// TwinCAT 3 PLC project Sample_Delivery
// ProgramVersion: 3.1.4023.0
// libraries:
//   lcls-twincat-sample-delivery, * (SLAC)
//   Tc2_Standard, * (Beckhoff Automation GmbH)
//   Tc2_System, * (Beckhoff Automation GmbH)
//   Tc3_Module, * (Beckhoff Automation GmbH)
// project tree:
//   / PlcTask.TcTTO
//   POUs/ MAIN.TcPOU
// real-time tasks:
//   TASK PlcTask: cycle T#10ms, priority 20, ADS port 350
// I/O:
//   DEVICE Device 1 (EtherCAT), AmsNetId 172.21.38.26.2.1
//     Term 1 (EK1200)
//     Box 3 (EP9128-0021) [EP9128-0021 8x EtherCAT junction]
//       Term 4 (EP9128-1021) [EP9128-1021 8x EtherCAT junction - Dev A]
//       Term 5 (EP9128-2021) [EP9128-2021 8x EtherCAT junction - Dev B]
//         Box 6 (EP1111)
//         M3 Selector A Digital IO (EP2338-1001)
//         M3 Selector A Serial IO (EP6002-0002)
// variable links:
//   Sample-Delivery Instance <-> Device 1 (EtherCAT)/Box 3 (EP9128-0021)/Term 5 (EP9128-2021)/M3 Selector A Digital IO (EP2338-1001)
//     PlcTask Outputs/MAIN.fbSelectorA.stShaker01.q_xPwrDO <-> Channel 9/Output
//     PlcTask Outputs/MAIN.fbSelectorA.stShaker02.q_xPwrDO <-> Channel 10/Output
//     PlcTask Outputs/MAIN.fbSelectorA.stShaker03.q_xPwrDO <-> Channel 11/Output
//     PlcTask Outputs/MAIN.fbSelectorA.stShaker04.q_xPwrDO <-> Channel 12/Output
//   Sample-Delivery Instance <-> Device 1 (EtherCAT)/Box 3 (EP9128-0021)/Term 5 (EP9128-2021)/M3 Selector A Serial IO (EP6002-0002)
//     PlcTask Inputs/MAIN.fbSelectorA.stSensSerial.stComIn/Status <-> COM TxPDO-Map Inputs Channel 1/Status
//     PlcTask Inputs/MAIN.fbSelectorA.stViciSerial.stComIn/Status <-> COM TxPDO-Map Inputs Channel 2/Status
//     PlcTask Outputs/MAIN.fbSelectorA.stSensSerial.stComOut/Ctrl <-> COM RxPDO-Map Outputs Channel 1/Ctrl
//     PlcTask Outputs/MAIN.fbSelectorA.stViciSerial.stComOut/Ctrl <-> COM RxPDO-Map Outputs Channel 2/Ctrl

CONFIGURATION Sample_Delivery
    RESOURCE PLC ON TwinCAT3
        TASK PlcTask(INTERVAL := T#10ms, PRIORITY := 20);
        PROGRAM MAIN WITH PlcTask : MAIN;
    END_RESOURCE
END_CONFIGURATION

// ---- POUs/MAIN.TcPOU
PROGRAM MAIN
VAR
	{attribute 'pytmc' := 'pv: TST:ICL:SEL:A'}
{attribute 'TcLinkTo' := '.stSensSerial.stComIn.Status := TIIB[M3 Selector A Serial IO (EP6002-0002)]^COM TxPDO-Map Inputs Channel 1^Status;
                          .stViciSerial.stComIn.Status := TIIB[M3 Selector A Serial IO (EP6002-0002)]^COM TxPDO-Map Inputs Channel 2^Status;
                          .stSensSerial.stComOut.Ctrl := TIID^Device 1 (EtherCAT)^Box 3 (EP9128-0021)^Term 5 (EP9128-2021)^M3 Selector A Serial IO (EP6002-0002)^COM RxPDO-Map Outputs Channel 1^Ctrl;
                          .stViciSerial.stComOut.Ctrl := TIID^Device 1 (EtherCAT)^Box 3 (EP9128-0021)^Term 5 (EP9128-2021)^M3 Selector A Serial IO (EP6002-0002)^COM RxPDO-Map Outputs Channel 2^Ctrl;
                          .stShaker01.q_xPwrDO := TIIB[M3 Selector A Digital IO (EP2338-1001)]^Channel 9^Output;
                          .stShaker02.q_xPwrDO := TIIB[M3 Selector A Digital IO (EP2338-1001)]^Channel 10^Output;
                          .stShaker03.q_xPwrDO := TIIB[M3 Selector A Digital IO (EP2338-1001)]^Channel 11^Output;
                          .stShaker04.q_xPwrDO := TIIB[M3 Selector A Digital IO (EP2338-1001)]^Channel 12^Output;
                          .stBaseIO.i_SyncUnitWC := TIID^MAIN (EtherCAT)^M3 Selector A (EP1111)^WcState^WcState;
'}
fbSelectorA : FB_SelectorM3;
END_VAR

fbSelectorA();

g_xFirstPass := FALSE;

END_PROGRAM
